{attribute 'qualified_only'}
{attribute 'strict'}
TYPE E_LTUHardwareState :
(
	NoCommand,
	RunForward,
	RunReverse,
	RunLeft,
	RunRight
);
END_TYPE

(* stored: Version 1.1.0.1, ProductVersion 3.1.4024.12
   DUT E_LTUHardwareState: Id {0b0806ee-50a7-4b02-85bb-3a011151da6a} *)
